# EPICS StreamDevice protocol: epics_installer_v1.0/option/serialTest_RAON_20220420/db/OBC.proto
ReplyTimeout = 200;
InTerminator = CR;
# No outTerminator because we need to send ENQ clean or RS485 will mess up the reply.

address = ESC "0\$1"; # for RS485

set2nominalspeed
{
    out "#\$1NSP" CR;
    in "#\$1,OK";
}

definespeedsetinstandby
{
    out "#\$1RPM,%05d" CR;
    in "#\$1,OK";
}

switchspeedsetpointtostandby
{
    out "#\$1SBY" CR;
    in "#\$1,OK";
}

set_rs232
{
    out "#\$1OPT14,2" CR;
    in "#\$1,OK";
}

set_onoff
{
    out "#\$1%{TMPOFF|TMPON}" CR;
    in  "#\$1,OK";
}

read_statusLEV
{
    out "#\$1LEV10" CR;
    in "#\$1,"
       "%(\$2:NOMINAL_SPEED_SET_POINT.A)d,"
       "%(\$2:STANDBY_SPEED_SET_POINT.A)d,"
       "00000,"
       "0,"
       "%(\$2:PUMP_RUNNING_TIME.A)d,"
       "%(\$2:ELECTRONIC_WORKING_TIME.A)d,"
       "00000,"
       "0000,"
       "0000,"
       "%(\$2:AT_SPEED_RELAY_THRESHOLD.A)d,"
       "%(\$2:CONTROL_TEMPERATURE.A)d,"
       "%(\$2:BEARING_THRESHOLD.A)d,"
       "%(\$2:BEARING_CURRENT_VALUE.A)d";
}

read_statusSTA
{
    out "#\$1STA" CR;
    in "#\$1,"
       "%(\$2:ORDER_STATUS.A)01r%(\$2:PUMP_STATUS.A)01r%(\$2:VALVE_STATUS.A)01r,"
       "%(\$2:CURRENT_SPEED.A)d,"
       "%(\$2:RADIAL_Yh.A)d,"
       "%(\$2:RADIAL_Xh.A)d,"
       "%(\$2:RADIAL_Yb.A)d,"
       "%(\$2:RADIAL_Xb.A)d,"
       "%(\$2:AXIAL_Z.A)d,"
       "%(\$2:MOTOR_CURRENT_VOLTAGE.A)d,"
       "%(\$2:MOTOR_CURRENT.A)d,"
       "%(\$2:PUMP_TEMP.A)d,"
       "%(\$2:CONTROLL_TEMP.A)d,"
       "%032d";
}

read_status
{
    read_statusLEV;
    read_statusSTA;
}
